# EPICS substitutions: soft_iocs/newport/iocBoot/iocnewport_d_hutch/XPSAux.substitutions
file "$(MOTOR)/db/XPSAuxLi.db"
{
pattern
{P,     R,          PORT,       CHAN,   SCAN}
{18ID_Newport_D:,  XPSAux1Li,  XPS_AUX1,   0,      "I/O Intr"}
{18ID_Newport_D:,  XPSAux2Li,  XPS_AUX1,   1,      "I/O Intr"}
{18ID_Newport_D:,  XPSAux3Li,  XPS_AUX1,   2,      "I/O Intr"}
{18ID_Newport_D:,  XPSAux4Li,  XPS_AUX1,   3,      "I/O Intr"}
}

file "$(MOTOR)/db/XPSAuxBi.db"
{
pattern
{P,    R,           PORT,     CHAN,  MASK,     SCAN}
{18ID_Newport_D:, XPSAux1Bi0,  XPS_AUX1, 0,     0x000001, "I/O Intr"}
{18ID_Newport_D:, XPSAux1Bi1,  XPS_AUX1, 0,     0x000002, "I/O Intr"}
{18ID_Newport_D:, XPSAux1Bi2,  XPS_AUX1, 0,     0x000004, "I/O Intr"}
{18ID_Newport_D:, XPSAux1Bi3,  XPS_AUX1, 0,     0x000008, "I/O Intr"}
{18ID_Newport_D:, XPSAux1Bi4,  XPS_AUX1, 0,     0x000010, "I/O Intr"}
{18ID_Newport_D:, XPSAux1Bi5,  XPS_AUX1, 0,     0x000020, "I/O Intr"}
{18ID_Newport_D:, XPSAux1Bi6,  XPS_AUX1, 0,     0x000040, "I/O Intr"}
{18ID_Newport_D:, XPSAux1Bi7,  XPS_AUX1, 0,     0x000080, "I/O Intr"}
{18ID_Newport_D:, XPSAux2Bi0,  XPS_AUX1, 1,     0x000001, "I/O Intr"}
{18ID_Newport_D:, XPSAux2Bi1,  XPS_AUX1, 1,     0x000002, "I/O Intr"}
{18ID_Newport_D:, XPSAux2Bi2,  XPS_AUX1, 1,     0x000004, "I/O Intr"}
{18ID_Newport_D:, XPSAux2Bi3,  XPS_AUX1, 1,     0x000008, "I/O Intr"}
{18ID_Newport_D:, XPSAux2Bi4,  XPS_AUX1, 1,     0x000010, "I/O Intr"}
{18ID_Newport_D:, XPSAux2Bi5,  XPS_AUX1, 1,     0x000020, "I/O Intr"}
{18ID_Newport_D:, XPSAux3Bi0,  XPS_AUX1, 2,     0x000001, "I/O Intr"}
{18ID_Newport_D:, XPSAux3Bi1,  XPS_AUX1, 2,     0x000002, "I/O Intr"}
{18ID_Newport_D:, XPSAux3Bi2,  XPS_AUX1, 2,     0x000004, "I/O Intr"}
{18ID_Newport_D:, XPSAux3Bi3,  XPS_AUX1, 2,     0x000008, "I/O Intr"}
{18ID_Newport_D:, XPSAux3Bi4,  XPS_AUX1, 2,     0x000010, "I/O Intr"}
{18ID_Newport_D:, XPSAux3Bi5,  XPS_AUX1, 2,     0x000020, "I/O Intr"}
{18ID_Newport_D:, XPSAux4Bi0,  XPS_AUX1, 3,     0x000001, "I/O Intr"}
{18ID_Newport_D:, XPSAux4Bi1,  XPS_AUX1, 3,     0x000002, "I/O Intr"}
{18ID_Newport_D:, XPSAux4Bi2,  XPS_AUX1, 3,     0x000004, "I/O Intr"}
{18ID_Newport_D:, XPSAux4Bi3,  XPS_AUX1, 3,     0x000008, "I/O Intr"}
{18ID_Newport_D:, XPSAux4Bi4,  XPS_AUX1, 3,     0x000010, "I/O Intr"}
{18ID_Newport_D:, XPSAux4Bi5,  XPS_AUX1, 3,     0x000020, "I/O Intr"}
{18ID_Newport_D:, XPSAux4Bi6,  XPS_AUX1, 3,     0x000040, "I/O Intr"}
{18ID_Newport_D:, XPSAux4Bi7,  XPS_AUX1, 3,     0x000080, "I/O Intr"}
{18ID_Newport_D:, XPSAux4Bi8,  XPS_AUX1, 3,     0x000100, "I/O Intr"}
{18ID_Newport_D:, XPSAux4Bi9,  XPS_AUX1, 3,     0x000200, "I/O Intr"}
{18ID_Newport_D:, XPSAux4Bi10, XPS_AUX1, 3,     0x000400, "I/O Intr"}
{18ID_Newport_D:, XPSAux4Bi11, XPS_AUX1, 3,     0x000800, "I/O Intr"}
{18ID_Newport_D:, XPSAux4Bi12, XPS_AUX1, 3,     0x001000, "I/O Intr"}
{18ID_Newport_D:, XPSAux4Bi13, XPS_AUX1, 3,     0x002000, "I/O Intr"}
{18ID_Newport_D:, XPSAux4Bi14, XPS_AUX1, 3,     0x004000, "I/O Intr"}
{18ID_Newport_D:, XPSAux4Bi15, XPS_AUX1, 3,     0x008000, "I/O Intr"}
}

file "$(MOTOR)/db/XPSAuxBo.db"
{
pattern
{P,    R,           PORT,     CHAN, MASK}
{18ID_Newport_D:, XPSAux1Bo0,  XPS_AUX1, 0,    0x000001}
{18ID_Newport_D:, XPSAux1Bo1,  XPS_AUX1, 0,    0x000002}
{18ID_Newport_D:, XPSAux1Bo2,  XPS_AUX1, 0,    0x000004}
{18ID_Newport_D:, XPSAux1Bo3,  XPS_AUX1, 0,    0x000008}
{18ID_Newport_D:, XPSAux1Bo4,  XPS_AUX1, 0,    0x000010}
{18ID_Newport_D:, XPSAux1Bo5,  XPS_AUX1, 0,    0x000020}
{18ID_Newport_D:, XPSAux1Bo6,  XPS_AUX1, 0,    0x000040}
{18ID_Newport_D:, XPSAux1Bo7,  XPS_AUX1, 0,    0x000080}
{18ID_Newport_D:, XPSAux3Bo0,  XPS_AUX1, 1,    0x000001}
{18ID_Newport_D:, XPSAux3Bo1,  XPS_AUX1, 1,    0x000002}
{18ID_Newport_D:, XPSAux3Bo2,  XPS_AUX1, 1,    0x000004}
{18ID_Newport_D:, XPSAux3Bo3,  XPS_AUX1, 1,    0x000008}
{18ID_Newport_D:, XPSAux3Bo4,  XPS_AUX1, 1,    0x000010}
{18ID_Newport_D:, XPSAux3Bo5,  XPS_AUX1, 1,    0x000020}
{18ID_Newport_D:, XPSAux4Bo0,  XPS_AUX1, 2,    0x000001}
{18ID_Newport_D:, XPSAux4Bo1,  XPS_AUX1, 2,    0x000002}
{18ID_Newport_D:, XPSAux4Bo2,  XPS_AUX1, 2,    0x000004}
{18ID_Newport_D:, XPSAux4Bo3,  XPS_AUX1, 2,    0x000008}
{18ID_Newport_D:, XPSAux4Bo4,  XPS_AUX1, 2,    0x000010}
{18ID_Newport_D:, XPSAux4Bo5,  XPS_AUX1, 2,    0x000020}
{18ID_Newport_D:, XPSAux4Bo6,  XPS_AUX1, 2,    0x000040}
{18ID_Newport_D:, XPSAux4Bo7,  XPS_AUX1, 2,    0x000080}
{18ID_Newport_D:, XPSAux4Bo8,  XPS_AUX1, 2,    0x000100}
{18ID_Newport_D:, XPSAux4Bo9,  XPS_AUX1, 2,    0x000200}
{18ID_Newport_D:, XPSAux4Bo10, XPS_AUX1, 2,    0x000400}
{18ID_Newport_D:, XPSAux4Bo11, XPS_AUX1, 2,    0x000800}
{18ID_Newport_D:, XPSAux4Bo12, XPS_AUX1, 2,    0x001000}
{18ID_Newport_D:, XPSAux4Bo13, XPS_AUX1, 2,    0x002000}
{18ID_Newport_D:, XPSAux4Bo14, XPS_AUX1, 2,    0x004000}
{18ID_Newport_D:, XPSAux4Bo15, XPS_AUX1, 2,    0x008000}
}

file "$(MOTOR)/db/XPSAuxLo.db"
{
pattern
{P,     R,         PORT,     CHAN}
{18ID_Newport_D:,  XPSAux1Lo, XPS_AUX1, 0}
{18ID_Newport_D:,  XPSAux3Lo, XPS_AUX1, 1}
{18ID_Newport_D:,  XPSAux4Lo, XPS_AUX1, 2}
}

file "$(MOTOR)/db/XPSAuxAi.db"
{
pattern
{P,    R,          PORT,     CHAN, LOPR,   HOPR,  PREC, SCAN}
{18ID_Newport_D:, XPSAuxAi0,  XPS_AUX1, 0,    -10.0,  10.0,  4,    "1 second"}
{18ID_Newport_D:, XPSAuxAi1,  XPS_AUX1, 1,    -10.0,  10.0,  4,    "1 second"}
{18ID_Newport_D:, XPSAuxAi2,  XPS_AUX1, 2,    -10.0,  10.0,  4,    "1 second"}
{18ID_Newport_D:, XPSAuxAi3,  XPS_AUX1, 3,    -10.0,  10.0,  4,    "1 second"}
}

file "$(MOTOR)/db/XPSAuxAo.db"
{
pattern
{P,    R,          PORT,     CHAN, DRVL,   LOPR,   DRVH,  HOPR,  PREC}
{18ID_Newport_D:, XPSAuxAo0,  XPS_AUX1, 0,    -10.0,  -10.0,  10.0,  10.0,   4}
{18ID_Newport_D:, XPSAuxAo1,  XPS_AUX1, 1,    -10.0,  -10.0,  10.0,  10.0,   4}
{18ID_Newport_D:, XPSAuxAo2,  XPS_AUX1, 2,    -10.0,  -10.0,  10.0,  10.0,   4}
{18ID_Newport_D:, XPSAuxAo3,  XPS_AUX1, 3,    -10.0,  -10.0,  10.0,  10.0    4}
}
